// TIA Portal V17 export
// export: Created 2023-11-27T22:24:51.2985434Z, ExportSetting WithDefaults, DisplayName Totally Integrated Automation Portal, DisplayVersion V17, DisplayName TIA Portal Openness, DisplayVersion V17, DisplayName TIA Portal Teamcenter Gateway, DisplayVersion V17, DisplayName TIA Portal Version Control Interface, DisplayVersion V17, DisplayName STEP 7 Professional, DisplayVersion V17, DisplayName STEP 7 Safety, DisplayVersion V17, DisplayName WinCC Advanced / Unified PC, DisplayVersion V17
DATA_BLOCK "V"   // DB4
{ S7_Optimized_Access := 'TRUE' }
VERSION : 0.1
// stored: AutoNumber true, IsOnlyStoredInLoadMemory false, IsWriteProtectedInAS false
   VAR
      _put_NW { S7_SetPoint := 'True'} : "sPut";
      _get { S7_SetPoint := 'True'} : "sGet";
      put_get { S7_SetPoint := 'True'} : Bool;
      put_get_prev_N : Bool;
      put_get_prev_P : Bool;
   END_VAR
BEGIN
END_DATA_BLOCK
